{attribute 'qualified_only'}
{attribute 'strict'}
{attribute 'to_string'}
TYPE eMessageTypes :
(
	HINT := 0,
	WARN := 1,
	ERROR := 2
	
);
END_TYPE

(* stored: Version 1.1.0.1, ProductVersion 3.1.4026.18
   DUT eMessageTypes: Id {8205eee8-71f6-48cb-9fd2-f10a91d2aa86} *)
